PROGRAM Version
VAR
END_VAR

//	版本号		修改人		修改日期		修改内容
//	1.2.0		李天		2021.06.27		311空跑后优化373解锁校平气缸
//	1.3.0		李天		2021.06.27		添加下工装阻挡气缸判断
//  1.4.0      刘雪峰       2021.06.28      添加下工装阻挡气缸屏蔽，优化气缸屏蔽，增加气缸空跑程序的调用选择
//  1.5.0      刘雪峰       2021.06.28      添加轴命名，添加取UC模组升降Z2气缸IO屏蔽，增加版本号界面显示，完善转向站和取uc模组流程，增加取uc模组z1z2气缸控制方法调用的判断,完善各机型气缸空跑程序
//  2.0.0      刘雪峰       2021.06.29      更新IO,气缸、轴excel,新增取UC工装夹紧气缸和IO,更新input和output结构体,更新E_cycliner枚举变量,按照机型屏蔽新增的气缸和IO,更新input和output的Textlist,优化取UC工站和取UC模组工站流程,完善正常模式下调用的A_Cylinder程序
//  2.1.0      刘雪峰       2021.07.01      更新气缸调试部分的界面程序，增加产品类型选择，优化转向站和下UC线体流程，添加取UC模组夹紧气缸工作位和解锁站侧推气缸2初始位在空跑时的屏蔽
//	2.2.0		李天		2021.07.02		修改373解锁校平气缸2动作,该气缸只需一直伸出即可;
//  2.2.1      刘雪峰       2021.07.05      修改部分气缸的界面调试控件，优化转向站初始化气缸动作流程；
//  2.3.0       王恒        2021.07.14      增加拨料站（Switch）和翻转站（Tipper）,将接驳模组拨料气缸和接驳模组升降气缸单独组成拨料站，将下UC皮带翻转气缸和下UC皮带顶升气缸单独组成翻转站;
//  2.3.1       王恒        2021.07.23      增加各工站到位光电检测超时报警;增加气缸界面按工站分页功能;主界面增加界面CT显示;增加生产计数显示;增加各到位光电信号显示;增加从转向站手动上料和从下UC、下工装皮带末端手动下料功能；增加屏蔽取UC模组功能，使投入工装时，只验证解锁与扣合，不验证夹取UC动作；
//                                          增加初始化检测各工站光电是否检测有料功能，并在初始化结束添加再次提醒操作员人工检查的5级报警;201机型下UC皮带流入光电IN6B代替下UC皮带翻转光电IN6D,用来检测UC是否到位，下UC皮带翻转光电IN6D不再使用；因为取UC模组Z1气缸上升速度较慢，所以下调了取UC模组Z1气缸的上限位，使Z1气缸的行程尽可能减少;
//  2.3.2       李天        2021.07.25      增加伺服轴持续接触极限报警，无法点动脱离问题，增加相应指示灯和复位功能；
//	2.4.0		李天		2021.07.26		将王恒新增的两个工站（接驳模组站及下UC线体旋转站） 再改回去
//	2.5.0		李天		2021.07.26		在RH069中待料测试 并修改一些细节 不影响整体流程
//	2.5.1		李天		2021.07.27		将手动下UC 手动下工装 手动上料 开放到界面
//	2.5.2		李天		2021.07.27		将报警显示控件放大
//	2.6.0		李天		2021.07.27		修改手动上料跳转空步号问题
//	2.6.1		李天		2021.07.28		添加用户权限 用户名：Admin 密码：333
//	2.6.2		李伟3		2021.07.28		优化201取UC站侧推气缸动作 可提前推出
//	2.7.0		李天		2021.07.31		将下UC流线及下工装流线到位光电报警等级改成3级
//	2.7.1		李伟3		2021.08.2		将自动流程中1471步中取UC模组平移Y气缸硬件IO修改为气缸功能块状态位
//	3.0.0		李伟3		2021.08.3		1.将自动流程中1471步中取UC模组平移Y气缸气缸功能块状态位修改为硬件IO
//                                          2.暂时取消手动页面权限管理，方便调试
//                                          3.将IO监控页面IN6B下工装线体流入光电变更为下工装流线流入光电
//                                          4.修改取UC模组自动程序，添加分支:设备机型为311时，取UC旋转气缸不旋转放料
//                                          5.将设备内工位检测到位光电传感器超时报警由五级报警提升为三级报警，并修复报警无法复位问题
//                                          6.添加 IN6F取UC模组平移Y气缸安全位 传感器,并修改动作流程
//                                          7.修改和优化了311机型设备 取UC站&取UC模组 的自动动作流程,缩短CT时间
//                                          8.在自动程序中添加 下UC线体到位检测超时 报警
//	3.0.1		李伟3		2021.08.5		1.屏蔽画面中添加屏蔽主流线分料气缸的功能
//                                          2.将主画面计数清零按钮增加用户权限
//                                          3.优化修改367机型 取UC模组 自动流程,缩短CT
//                                          4.优化画面按钮相关中文显示
//                                          5.修复了下工装站初始化撞机的问题
//	3.0.2		李伟3		2021.08.6		1.屏蔽画面中添加 蜂鸣器屏蔽 和 安全门屏蔽 的功能
//                                          2.增加 设备运行中安全门被打开 报警
//	4.0.0		李伟3		2021.08.12		1.373机型解锁站增加两个气缸，增加手动&自动&初始化程序
//                                          2.修复373机型手动画面校平气缸未屏蔽的问题
//                                          3.修复373机型IO画面未使用IO点没有屏蔽的问题
//                                          4.修复设备蜂鸣器响声不正常的问题
//                                          5.优化367机型取UC站的自动流程
//	4.1.0		李伟3		2021.08.13		1.增加接驳线阻挡气缸&接驳线光电传感器，增加手动&自动&初始化程序
//	4.1.1		李伟3		2021.08.16		1.优化不同机型手动页面&IO监控页面的显示问题
//	4.2.0		李伟3		2021.08.24		1.将新加的接驳站前流水线由急停按钮控制改为继电器控制，增加手自动程序
//	4.2.1		李伟3		2021.08.25		1.优化201机型下UC皮带翻转顶升气缸动作流程，先让顶升气缸上升再放UC，防止损伤排线
//	4.2.2		李伟3		2021.08.31		1.优化主流线分料气缸和阻挡气缸的动作逻辑,修改主流线分料气缸缩回端为原位,增加主流线阻挡光电检测超时报警
//	4.3.0		李伟3		2021.09.02		1.367机型增加主流线拨料升降气缸，修改手自动程序及画面
//                                          2.修改取UC站初始化动作流程，修复367机型取UC站初始化异常的问题
//	5.0.0		李伟3		2021.09.07		1.增加通过EIP与前站信号交互的配置和程序
//                                          2.修改主流线到位光电检测超时时间为20S,因为主流线速度过慢会误引发报警
//	5.1.0		李伟3		2021.09.10		1.优化了主流线和接驳线上料优先级选择部分的程序，画面上增加了优先级下拉菜单选择
//                                          2.画面上增加了停止前站放料的按钮
//                                          3.增加 主流线拨料气缸安全位 IN0C 传感器，优化367主流线上料流程
//                                          4.增加主流线与接驳线上料优先级根据传感器自动切换逻辑
//                                          5.优化与前站交互要料逻辑
//	5.2.0		李伟3		2021.09.16		1.311机型增加检测工装误合盖传感器，修改动作流程及画面
//                                          2.367机型增加解锁站流入光电传感器，优化动作流程，缩短CT
//                                          3.373机型增加取UC站流入光电传感器，优化动作流程，缩短CT
//                                          4.373机型增加主流线传感器,优化367机型主流线拨料气缸动作，增加主流线拨料升降气缸上升速度过慢报警，防止损伤产品
//                                          5.优化自动程序中所使用的延时，画面上增加延时时间设置
//                                          6.将打开安全门由一级报警修改为3级报警，方便维护
//                                          7.修复取UC站初始化时与取UC模组撞机的问题
//	5.3.0		李伟3		2021.09.17		1.373机型取UC站增加检测工装误合盖传感器，修改动作流程及画面
//	5.4.0		李伟3		2021.09.17		1.修改解锁站和取UC站的放料逻辑，缩短CT
//	5.5.0		李伟3		2021.09.17		1.将接驳站分料气缸和阻挡气缸分离为单独工站，优化交互逻辑

END_PROGRAM

(* stored: Version 1.1.0.1, ProductVersion 3.1.4024.3
   POU Version: Id {e7afc2a9-56be-44f0-a4b7-0bdfa935308f}, SpecialFunc None *)
